TYPE RotatingSwitchConfigs :
STRUCT
	ELL18RotatingSwitchConfig : ELL18AttenuationFilterConfig;
END_STRUCT
END_TYPE

(* stored: Version 1.1.0.1, ProductVersion 3.1.4024.10
   DUT RotatingSwitchConfigs: Id {891c257a-2867-4327-8d53-efbbcdd9ed6a} *)
